// TIA Portal V16 export
// export: Created 2022-09-01T14:27:09.6689539Z, ExportSetting WithDefaults, DisplayName Totally Integrated Automation Portal, DisplayVersion V16, DisplayName TIA Portal Version Control Interface, DisplayVersion V16, DisplayName TIA Portal Openness, DisplayVersion V16, DisplayName STEP 7 Professional, DisplayVersion V16, DisplayName STEP 7 Safety, DisplayVersion V16, DisplayName WinCC Advanced, DisplayVersion V16
VAR_GLOBAL   // PLC tag table "Outputs"
   "EV1.1" AT %Q0.0 : Bool;
   "EV2.1" AT %Q0.1 : Bool;
   "EV3.1" AT %Q0.2 : Bool;
   "EV4.1" AT %Q0.3 : Bool;
   "EV5.1" AT %Q0.4 : Bool;
   "EV1.2" AT %Q0.5 : Bool;
   "EV2.2" AT %Q0.6 : Bool;
   "EV3.2" AT %Q0.7 : Bool;
   "EV4.2" AT %Q1.0 : Bool;
   "EV5.2" AT %Q1.1 : Bool;
   BOMBA_1_VAR AT %Q2.0 : Bool;
   BOMBA_2_VAR AT %Q2.1 : Bool;
   BOMBA_3_RESERVA AT %Q2.2 : Bool;
   ULTRAVIOLETA AT %Q2.3 : Bool;
END_VAR
